FUNCTION_BLOCK fbIO_AnalogueInput
VAR_INPUT
	iInMode:		INT;
	iInValue:		INT;
	iInSensorType:	INT;
	rInEngUnitsMin:	REAL;
	rInEngUnitsMax:	REAL;
	rInLowLow:		REAL;
	rInLow:			REAL;
	rInHigh:		REAL;
	rInHighHigh:	REAL;
	rInLowLowDeadband: REAL;
	rInLowDeadband:REAL;
	rInHighDeadband:REAL;
	rInHighHighDeadband:REAL;
	bInResetError:BOOL;
END_VAR
VAR_OUTPUT
	rOutEngUnitsValue:REAL; (*Engineering units scaled value*)
	bOutLowLow:BOOL; (*Low low alarm is active*)
	bOutLow:BOOL; (*Low warning is active*)
	bOutHigh:BOOL; (*High warning is active*)
	bOutHighHigh:BOOL; (*High high alarm is active*)
	bOutAuto:BOOL; (*Input is in auto mode*)
	bOutError:BOOL; (*Error Exists*)
	ERROR_IO_AnalogueIn:stError_AnalogueInput;
END_VAR

VAR_IN_OUT
	HMI_IO_AnalogueInput:stHMI_AnalogueInput;
END_VAR

VAR
	fScaled16:REAL;
	fTempScaled16:REAL;
	ftempScaled16_a:REAL;
	ftempScaled16_b:REAL;
	bTest:BOOL;
END_VAR

//Process Alarms limits
bOutLowLow:= (rOutEngUnitsValue<=(rInLowLow-rInLowLowDeadband));  	// LL Alarm
bOutLow:= (rOutEngUnitsValue<=(rInLow-rInLowDeadband));  			// LL Warning
bOutHighHigh:= (rOutEngUnitsValue>=(rInHigh+rInHighHighDeadband));  	// HH Alarm	
bOutHigh:= (rOutEngUnitsValue>=(rInHighHigh+rInHighDeadband));  		// HH Warning	
	
bOutAuto := iInMode=1;

(***************************SCALING ANALOGUE************************
ftempScaled16_a:=
ftempScaled16_b:=
IF fTempScaled32 THEN
	
END_IF
*)

CASE iInMode OF
	0:
		;
	1:	// Auto mode
		rOutEngUnitsValue:=fScaled16;
	2:	// Manual Mode
		rOutEngUnitsValue:=HMI_IO_AnalogueInput.rManualValue;
		
	3:	// Independant
	END_CASE
	
(*Map Error bits*)
ERROR_IO_AnalogueIn.LowLowAlarm:=bOutLowLow;			//HH alarm
ERROR_IO_AnalogueIn.HighHighAlarm:=bOutHighHigh;		//LL Alarm	
	
(*map active value to the scada*)
HMI_IO_AnalogueInput.rInputValue:=fScaled16;
HMI_IO_AnalogueInput.rActiveValue:=rOutEngUnitsValue;

(*Error Code*)
HMI_IO_AnalogueInput.iErrorCode.0:=ERROR_IO_AnalogueIn.LowLowAlarm;	
HMI_IO_AnalogueInput.iErrorCode.1:=ERROR_IO_AnalogueIn.HighHighAlarm;	
HMI_IO_AnalogueInput.iErrorCode.2:=ERROR_IO_AnalogueIn.LowLowAlarm;	
HMI_IO_AnalogueInput.iErrorCode.3:=bTest;
	
HMI_IO_AnalogueInput.bError:=(HMI_IO_AnalogueInput.iErrorCode<>0);

END_FUNCTION_BLOCK

(* stored: Version 1.1.0.1, ProductVersion 3.1.4024.11
   POU fbIO_AnalogueInput: Id {805e4ee0-1d54-44f1-bb8f-ec68bf186558}, SpecialFunc None *)
